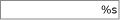
VISUALIZATION visSHOWDATA_QUERRY  // 120x20
VAR_INPUT
    visfbDATATYPEIn     :   ITF_DATATYPE;	
END_VAR
VAR_INPUT 
    stPhysikalischeEinheit  : STRING[5];
END_VAR
    Frame (0,0 120x20), invisible if: NOT __QUERYINTERFACE(visfbDATATYPEIn,visfbDATATYPEIn)
        shows visSHOWDATA_ITF(visfbDATATYPEIn := visfbDATATYPEIn, stPhysikalischeEinheit := stPhysikalischeEinheit)
END_VISUALIZATION

// 40 Visualizations/32 Bit/TIME/visTIME_ITF
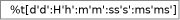
VISUALIZATION visTIME_ITF  // 180x20
VAR_INPUT
    visfbTIME   :   ITF_TIME;	
END_VAR
    Textfield (0,0 180x20), "%t[d'd':H'h':m'm':ss's':ms'ms']", text variable: visfbTIME.proValue
        OnMouseClick: write the text variable via InputWithLimits, min TO_UDINT(visfbTIME.proMin), max TO_UDINT(visfbTIME.proMax), title 'T#'
END_VISUALIZATION

// 40 Visualizations/32 Bit/TOD/visTOD
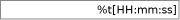
VISUALIZATION visTOD  // 180x20
VAR_INPUT   
    visfbTODIn :   ITF_DATATYPE;	
END_VAR
VAR  
    visfbTOD   :   ITF_TOD;	
END_VAR
    Frame (0,0 180x20), invisible if: NOT __QUERYINTERFACE(visfbTODIn,visfbTOD)
        shows visTOD_QUERRY(visfbTODIn := visfbTOD)
        pReferences[0]: visfbDATE_AND_TIMEIn=visfbTOD
END_VISUALIZATION

// 40 Visualizations/32 Bit/TIME/visTIME_QUERRY
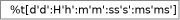
VISUALIZATION visTIME_QUERRY  // 180x20
VAR_INPUT
    visfbTIMEIn :   ITF_TIME;	
END_VAR
    Frame (0,0 180x20), invisible if: NOT __QUERYINTERFACE(visfbTIMEIn,visfbTIMEIn)
        shows visTIME_ITF(visfbTIME := visfbTIMEIn)
END_VISUALIZATION

// 40 Visualizations/16 Bit/INT/visINT_QUERRY
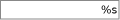
VISUALIZATION visINT_QUERRY  // 120x20
VAR_INPUT
    visfbINTIn :   ITF_INT;	
END_VAR
VAR_INPUT 
    stPhysikalischeEinheit  : STRING[5];
END_VAR
    Frame (0,0 120x20), invisible if: NOT __QUERYINTERFACE(visfbINTIn,visfbINTIn)
        shows visINT_ITF(visfbINT := visfbINTIn, stPhysikalischeEinheit := stPhysikalischeEinheit)
END_VISUALIZATION

// 40 Visualizations/32 Bit/DATE AND TIME/visDATE_AND_TIME
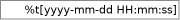
VISUALIZATION visDATE_AND_TIME  // 180x20
VAR_INPUT   
    visfbDATE_AND_TIMEIn :   ITF_DATATYPE;	
END_VAR
VAR  
    visfbDATE_AND_TIME   :   ITF_DATE_AND_TIME;	
END_VAR
    Frame (0,0 180x20), invisible if: NOT __QUERYINTERFACE(visfbDATE_AND_TIMEIn,visfbDATE_AND_TIME)
        shows visDATE_AND_TIME_QUERRY(visfbDATE_AND_TIMEIn := visfbDATE_AND_TIME)
END_VISUALIZATION

// 40 Visualizations/Show Data/visSHOWDATA
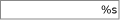
VISUALIZATION visSHOWDATA  // 120x20
VAR_INPUT
    visfbDATATYPEIn     :   ITF_DATATYPE;	
END_VAR
VAR
    visfbDATATYPE       :   ITF_DATATYPE;	
END_VAR
VAR_INPUT 
    stPhysikalischeEinheit  : STRING[5];
END_VAR
    Frame (0,0 120x20), invisible if: NOT __QUERYINTERFACE(visfbDATATYPEIn,visfbDATATYPE)
        shows visSHOWDATA_QUERRY(visfbDATATYPEIn := visfbDATATYPE, stPhysikalischeEinheit := stPhysikalischeEinheit)
END_VISUALIZATION

// 40 Visualizations/8 Bit/SINT/visSINT_ITF
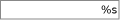
VISUALIZATION visSINT_ITF  // 120x20
VAR_INPUT
    visfbSINT   :   ITF_SINT;	
END_VAR
VAR_INPUT 
    stPhysikalischeEinheit  : STRING[5];
END_VAR
    Textfield (0,0 120x20), "%s", text variable: CONCAT(TO_STRING(visfbSINT.proValue),stPhysikalischeEinheit)
        OnMouseClick: write visfbSINT.proValue via InputWithLimits, min visfbSINT.proMin, max visfbSINT.proMax
END_VISUALIZATION

// 40 Visualizations/ENUMERATION/16 Bit/visENUMERATION_INT
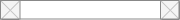
VISUALIZATION visENUMERATION_INT  // 180x20
VAR_INPUT
    visfbINT   :   ITF_INT;		
END_VAR
    Image (160,0 20x20), image: CtaVisSymbols.ImagePool.arrow-right_square
        OnMouseClick: execute {
            IF visfbINT.proValue < visfbINT.proMax THEN
                visfbINT.proValue := visfbINT.proValue + 1;
            ELSIF visfbINT.proValue = visfbINT.proMax THEN
                visfbINT.proValue := visfbINT.proMin;
            END_IF;
        }
    Image (0,0 20x20), image: CtaVisSymbols.ImagePool.arrow-left_square
        OnMouseClick: execute {
            IF visfbINT.proValue > visfbINT.proMin THEN
                visfbINT.proValue := visfbINT.proValue - 1;
            ELSIF visfbINT.proValue = visfbINT.proMin THEN
                visfbINT.proValue := visfbINT.proMax;
            END_IF;
        }
END_VISUALIZATION

// 40 Visualizations/8 Bit/BYTE/visBYTE_ITF
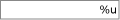
VISUALIZATION visBYTE_ITF  // 120x20
VAR_INPUT
    visfbBYTE   :   ITF_BYTE;	
END_VAR
    Textfield (0,0 120x20), "%u", text variable: visfbBYTE.proValue
        OnMouseClick: write the text variable via InputWithLimits, min visfbBYTE.proMin, max visfbBYTE.proMax
END_VISUALIZATION

// 40 Visualizations/32 Bit/TOD/visTOD_QUERRY
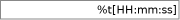
VISUALIZATION visTOD_QUERRY  // 180x20
VAR_INPUT
    visfbTODIn :   ITF_TOD;	
END_VAR
    Frame (0,0 180x20), invisible if: NOT __QUERYINTERFACE(visfbTODIn,visfbTODIn)
        shows visTOD_ITF(visfbTODIn := visfbTODIn)
END_VISUALIZATION

// 40 Visualizations/16 Bit/WORD/WORD HEX/visWORD_QUERRY_HEX
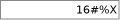
VISUALIZATION visWORD_QUERRY_HEX  // 120x20
VAR_INPUT
    visfbWORDIn :   ITF_WORD;	
END_VAR
    Frame (0,0 120x20), invisible if: NOT __QUERYINTERFACE(visfbWORDIn,visfbWORDIn)
        shows visWORD_ITF_HEX(visfbWORD := visfbWORDIn)
END_VISUALIZATION

// 40 Visualizations/ENUMERATION/visENUMERATION
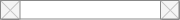
VISUALIZATION visENUMERATION  // 180x20
VAR_INPUT
    visfbENUIn :   ITF_DATATYPE;	
END_VAR
VAR
	visfbBYTE  :   ITF_BYTE;	
    visfbINT   :   ITF_INT;	
    visfbDINT  :   ITF_DINT;
END_VAR
    Rectangle (0,0 179x19)
    Frame (0,0 180x20), invisible if: NOT __QUERYINTERFACE(visfbENUIn,visfbINT)
        shows visENUMERATION_INT_QUERRY(visfbINT := visfbINT)
    Frame (0,0 180x20), invisible if: NOT __QUERYINTERFACE(visfbENUIn,visfbDINT)
        shows visENUMERATION_DINT_QUERRY(visfbDINT := visfbDINT)
    Frame (0,0 180x20), invisible if: NOT __QUERYINTERFACE(visfbENUIn,visfbBYTE)
        shows visENUMERATION_BYTE_QUERR(visfbBYTE := visfbBYTE)
END_VISUALIZATION

// 40 Visualizations/32 Bit/DINT/visDINT_QUERRY
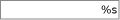
VISUALIZATION visDINT_QUERRY  // 120x20
VAR_INPUT
    visfbDINTIn :   ITF_DINT;	
END_VAR
VAR_INPUT 
    stPhysikalischeEinheit  : STRING[5];
END_VAR
    Frame (0,0 120x20), invisible if: NOT __QUERYINTERFACE(visfbDINTIn,visfbDINTIn)
        shows visDINT_ITF(visfbDINT := visfbDINTIn, stPhysikalischeEinheit := stPhysikalischeEinheit)
END_VISUALIZATION

// 40 Visualizations/16 Bit/UINT/visUINT
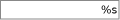
VISUALIZATION visUINT  // 120x20
VAR_INPUT
    visfbUINTIn :   ITF_DATATYPE;	
END_VAR
VAR
    visfbUINT   :   ITF_UINT;	
END_VAR
VAR_INPUT 
    stPhysikalischeEinheit  : STRING[5];
END_VAR
    Frame (0,0 120x20), invisible if: NOT __QUERYINTERFACE(visfbUINTIn,visfbUINT)
        shows visUINT_QUERRY(visfbUINTIn := visfbUINT, stPhysikalischeEinheit := stPhysikalischeEinheit)
END_VISUALIZATION

// 40 Visualizations/8 Bit/BYTE/visBYTE
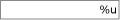
VISUALIZATION visBYTE  // 120x20
VAR_INPUT
    visfbBYTEIn  : ITF_DATATYPE;
END_VAR
VAR
    visfbBYTE   :   ITF_BYTE;	
END_VAR
    Frame (0,0 120x20), invisible if: NOT __QUERYINTERFACE(visfbBYTEIn,visfbBYTE)
        shows visBYTE_QUERRY(visfbBYTEIn := visfbBYTE)
END_VISUALIZATION

// 40 Visualizations/40 Byte String/visSTRING40_ITF
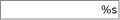
VISUALIZATION visSTRING40_ITF  // 120x20
VAR_INPUT
    visfbSTRING40In   :   ITF_STRING40;	
END_VAR
    Textfield (0,0 120x20), "%s", text variable: visfbSTRING40In.proValue
        OnMouseClick: write the text variable via Default
END_VISUALIZATION

// 40 Visualizations/ENUMERATION/16 Bit/visENUMERATION_INT_QUERRY
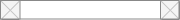
VISUALIZATION visENUMERATION_INT_QUERRY  // 180x20
VAR_INPUT
    visfbINT   :   ITF_INT;	
END_VAR
    Frame (0,0 180x20), invisible if: NOT __QUERYINTERFACE(visfbINT,visfbINT)
        shows visENUMERATION_INT(visfbINT := visfbINT)
END_VISUALIZATION

// 40 Visualizations/32 Bit/DINT/visDINT
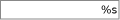
VISUALIZATION visDINT  // 120x20
VAR_INPUT
    visfbDINTIn :   ITF_DATATYPE;	
END_VAR
VAR
    visfbDINT   :   ITF_DINT;	
END_VAR
VAR_INPUT 
    stPhysikalischeEinheit  : STRING[5];
END_VAR
    Frame (0,0 120x20), invisible if: NOT __QUERYINTERFACE(visfbDINTIn,visfbDINT)
        shows visDINT_QUERRY(visfbDINTIn := visfbDINT, stPhysikalischeEinheit := stPhysikalischeEinheit)
END_VISUALIZATION

// 40 Visualizations/32 Bit/DATE AND TIME/visDATE_AND_TIME_QUERRY
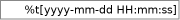
VISUALIZATION visDATE_AND_TIME_QUERRY  // 180x20
VAR_INPUT
    visfbDATE_AND_TIMEIn :   ITF_DATE_AND_TIME;	
END_VAR
    Frame (0,0 180x20), invisible if: NOT __QUERYINTERFACE(visfbDATE_AND_TIMEIn,visfbDATE_AND_TIMEIn)
        shows visDATE_AND_TIME_ITF(visfbDATE_AND_TIMEIn := visfbDATE_AND_TIMEIn)
END_VISUALIZATION

// 40 Visualizations/1 Bit/visBOOL_QUERRY
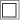
VISUALIZATION visBOOL_QUERRY  // 20x20
VAR_INPUT
    visfbBOOLIn  : ITF_BOOL;
END_VAR
    Frame (0,0 20x20), invisible if: NOT __QUERYINTERFACE(visfbBOOLIn,visfbBOOLIn)
        shows visBOOL_ITF(visfbBOOL := visfbBOOLIn)
END_VISUALIZATION

// 40 Visualizations/ENUMERATION/32 Bit/visENUMERATION_DINT
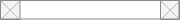
VISUALIZATION visENUMERATION_DINT  // 180x20
VAR_INPUT
    visfbDINT  :   ITF_DINT;		
END_VAR
    Image (160,0 20x20), image: CtaVisSymbols.ImagePool.arrow-right_square
        OnMouseClick: execute {
            IF visfbDINT.proValue < visfbDINT.proMax THEN
                visfbDINT.proValue := visfbDINT.proValue + 1;
            ELSE
                visfbDINT.proValue := visfbDINT.proMin;
            END_IF;
        }
    Image (0,0 20x20), image: CtaVisSymbols.ImagePool.arrow-left_square
        OnMouseClick: execute {
            IF visfbDINT.proValue > visfbDINT.proMin THEN
                visfbDINT.proValue := visfbDINT.proValue - 1;
            ELSE
                visfbDINT.proValue := visfbDINT.proMax;
            END_IF;
        }
END_VISUALIZATION

// 40 Visualizations/32 Bit/DINT/visDINT_ITF
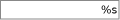
VISUALIZATION visDINT_ITF  // 120x20
VAR_INPUT
    visfbDINT   :   ITF_DINT;	
END_VAR
VAR_INPUT 
    stPhysikalischeEinheit  : STRING[5];
END_VAR
    Textfield (0,0 120x20), "%s", text variable: CONCAT(TO_STRING(visfbDINT.proValue),stPhysikalischeEinheit)
        OnMouseClick: write visfbDINT.proValue via InputWithLimits, min visfbDINT.proMin, max visfbDINT.proMax
END_VISUALIZATION

// 40 Visualizations/16 Bit/UINT/visUINT_ITF
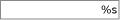
VISUALIZATION visUINT_ITF  // 120x20
VAR_INPUT
    visfbUINT   :   ITF_UINT;	
END_VAR
VAR_INPUT 
    stPhysikalischeEinheit  : STRING[5];
END_VAR
    Textfield (0,0 120x20), "%s", text variable: CONCAT(TO_STRING(visfbUINT.proValue),stPhysikalischeEinheit)
        OnMouseClick: write visfbUINT.proValue via InputWithLimits, min visfbUINT.proMin, max visfbUINT.proMax
END_VISUALIZATION

// 40 Visualizations/16 Bit/UINT/visUINT_QUERRY
